ADAPTER IOpCdtItems (* Adapter Interface *)
  (* Standard: 61499-1 *)
  (* Version 0.0, 6/5/2026, Schneider Electric *)
  PACKAGE SE.Nereda;
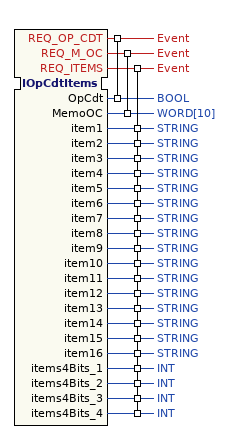
  EVENT_OUTPUT
    REQ_OP_CDT WITH OpCdt;
    REQ_M_OC WITH MemoOC;
    REQ_ITEMS WITH item1, item2, item3, item4, item5, item6, item7, item8, items4Bits_1, items4Bits_2, items4Bits_3, items4Bits_4, item9, item10, item11, item12, item13, item14, item15, item16;
  END_EVENT
  VAR_OUTPUT
    OpCdt : BOOL;
    MemoOC : ARRAY [0..9] OF WORD;
    item1 : STRING;
    item2 : STRING;
    item3 : STRING;
    item4 : STRING;
    item5 : STRING;
    item6 : STRING;
    item7 : STRING;
    item8 : STRING;
    item9 : STRING;
    item10 : STRING;
    item11 : STRING;
    item12 : STRING;
    item13 : STRING;
    item14 : STRING;
    item15 : STRING;
    item16 : STRING;
    items4Bits_1 : INT;
    items4Bits_2 : INT;
    items4Bits_3 : INT;
    items4Bits_4 : INT;
  END_VAR
  SERVICE SOCKET/PLUG
    SEQUENCE request_confirm
      SOCKET.REQ(REQD) -> PLUG.REQ(REQD);
      PLUG.CNF(CNFD) -> SOCKET.CNF(CNFD);
    END_SEQUENCE
    SEQUENCE indication_response
      PLUG.IND(INDD) -> SOCKET.IND(INDD);
      SOCKET.RSP(RSPD) -> PLUG.RSP(RSPD);
    END_SEQUENCE
  END_SERVICE
END_ADAPTER
